// TIA Portal V19 export
TYPE "EH_ProMag300_PD_UDT"
   STRUCT
      Addr : Int;   // First Byte address of 35 byte address space
      Totaliser_Mode : Byte;   // Configuration variable
      Volume_Flow : Real;   // Measured value: floating point number
      Actual_Diagnostics : Int;   // Diagnostic information number
      Totaliser_Value : Real;   // Measured value: floating point number
      Device_Status_VF : Byte;   // Status Code Hex Value
      Device_Status_AD : Byte;   // Status Code Hex Value
      Device_Status_TV : Byte;   // Status Code Hex Value
      Totaliser_Control : Byte;   // Control variable
   END_STRUCT;
END_TYPE
